# EPICS autosave request: iocBoot/ioc13idd/auto_positions_xps.req
file "CARS_motor_positions.req",         P=$(P), M=m81
file "CARS_motor_positions.req",         P=$(P), M=m82
file "CARS_motor_positions.req",         P=$(P), M=m83
file "CARS_motor_positions.req",         P=$(P), M=m84
